{attribute 'GeneratedUsingTerminal: EP1816-0008-0018'}
{attribute addProperty BoxType "EP1816-0008-0018"}
{attribute addProperty Id "DIG_Inputs_Channel_1AT %I*DIG_Inputs_Channel_CC4551489DIG_Inputs_Channel_2AT %I*DIG_Inputs_Channel_CC4551489WcStateAT %I*WcState_9091E0EB2InfoDataAT %I*InfoData_94A18F5E2"}
{attribute addProperty CRC "3864417421"}
{attribute addProperty Size "22"}
TYPE EP1816_E656548D EXTENDS EtcSlaveTerminalBase_947E5A46 :
STRUCT
	{attribute addProperty Name "DIG_Inputs_Channel_1"}
	DIG_Inputs_Channel_1 : DIG_Inputs_Channel_CC455148;
	{attribute addProperty Name "DIG_Inputs_Channel_2"}
	DIG_Inputs_Channel_2 : DIG_Inputs_Channel_CC455148;
	{attribute addProperty Name "WcState"}
	WcState : WcState_9091E0EB;
	{attribute addProperty Name "InfoData"}
	InfoData : InfoData_94A18F5E;
END_STRUCT
END_TYPE

(* stored: Version 1.2.0.0, ProductVersion 3.1.4024.9
   DUT EP1816_E656548D: Id {43c8c759-a8ff-4269-a80f-75b1255c5b58} *)
